TYPE ST_Xbox_NC_Halt_Dynamics :
STRUCT
	// Deceleration of the MC_Halt command
	fDeceleration : LREAL := 5000; 
	// Jerk of the MC_Halt command
    fJerk         : LREAL := 10000;
	// BufferMode of the MC_Halt command
    mcBufferMode   : MC_BufferMode; 
	// Options oif the MC_Halt command
    stOptions      : ST_MoveOptions; 
END_STRUCT
END_TYPE

(* stored: Version 1.1.0.1, ProductVersion 3.1.4024.11
   DUT ST_Xbox_NC_Halt_Dynamics: Id {22ef05d6-5e67-08ad-2b7b-8b4ec878a171} *)
